FUNCTION_BLOCK AxisReferencing
VAR_IN_OUT
	ReferenceSwitch:BOOL;
	AxisPlus:BOOL;
	AxisMinus:BOOL;
	Control:INT;
	SpeedPWM:INT;
	SetCounter:BOOL;
END_VAR
VAR_OUTPUT
	ReferenceOkay:BOOL;
END_VAR
VAR
END_VAR

IF ReferenceSwitch THEN
	AxisMinus := FALSE;
	AxisPlus := FALSE;
	Control := 0;
	SpeedPWM := 0;
	SetCounter := TRUE;
	ReferenceOkay:= TRUE;
ELSE
	AxisMinus := TRUE;
	AxisPlus := FALSE;
	Control := 32;
	SpeedPWM := 5000;
	SetCounter := FALSE;
END_IF

END_FUNCTION_BLOCK

(* stored: Version 1.1.0.1, ProductVersion 3.1.4024.12
   POU AxisReferencing: Id {30ee3797-0995-4380-9d12-6ee2c022fb21}, SpecialFunc None *)
